// TIA Portal V17 export
// export: Created 2025-03-10T13:12:01.4867511Z, ExportSetting WithDefaults, DisplayName Totally Integrated Automation Portal, DisplayVersion V17 Update 8, DisplayName TIA Portal Openness, DisplayVersion V17 Update 8, DisplayName TIA Portal Version Control Interface, DisplayVersion V17, DisplayName SINAMICS Startdrive Advanced, DisplayVersion V17 SP2, DisplayName SINAMICS Startdrive G110M, G120, G120C, G120D, G120P, G115D, DisplayVersion V17 SP2, DisplayName SINAMICS Startdrive G130, G150, S120, S150, SINAMICS MV, S210, DisplayVersion V17 SP2, DisplayName STEP 7 Professional, DisplayVersion V17 Update 8, DisplayName SINUMERIK ONE STEP 7 Toolbox, DisplayVersion V17 Update 12, DisplayName SINUMERIK 840D sl STEP 7 Toolbox, DisplayVersion V17 Update 12, DisplayName STEP 7 Safety, DisplayVersion V17 Update 6, DisplayName WinCC Advanced, DisplayVersion V17 Update 8
TYPE "LBP_typePowerrideConfigPos"
TITLE = Data type for configuration of a Powerride position / Tipo de datos para configurar una posición de powerride / Datentyp für Konfiguration einer Powerride Position
// User data type for LBP_PowerrideConfig (sub type) / Tipo de datos de usuario para LBP_PowerrideConfig (subtipo) / Anwenderdatentyp für LBP_PowerrideConfig (Untertyp)
// stored: IsFailsafeCompliant false
   STRUCT
      value { S7_SetPoint := 'True'} : USInt;   // Override-Faktor / override factor / Factor de corrección
      ledColor { S7_SetPoint := 'True'} : USInt;   // Farbe des LED-Bandes / color of scale LEDs / Color de la franja de LED
      vibrationIndex { S7_SetPoint := 'True'} : USInt;   // Index des Vibrationsmusters / index of vibration pattern / Índice de la plantilla de vibración
   END_STRUCT;
END_TYPE
